RoboDK station: first test.rdk

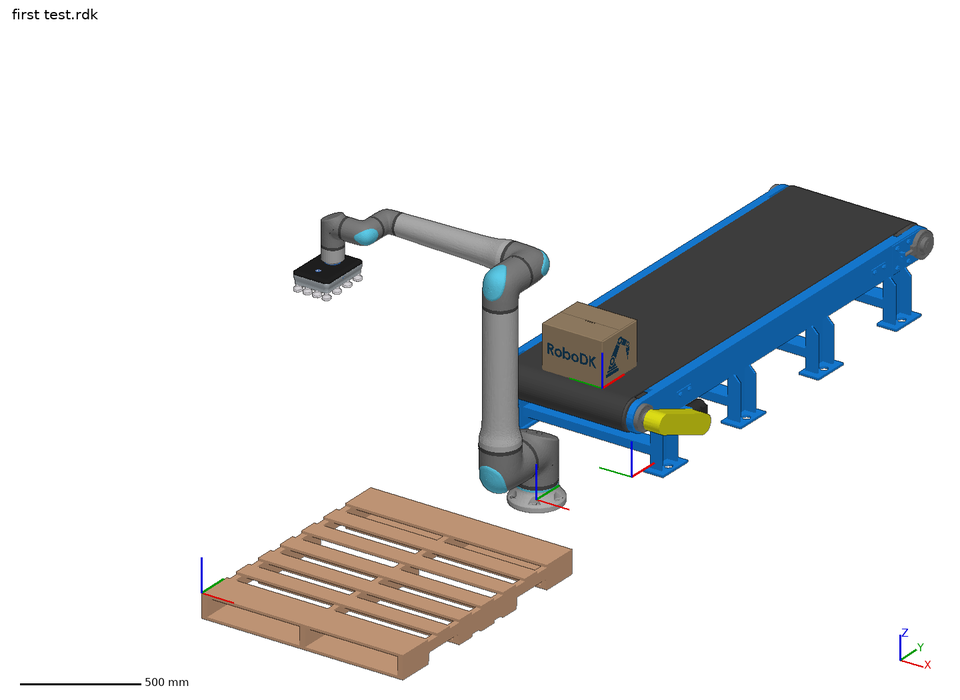
[picture v0: the station drawn from its stored meshes, robots at their saved joint values, targets as dots, program paths as lines]
Station first test (saved by RoboDK 5.9.2). Poses are relative to the parent item; angles as X-Y-Z fixed-axis rotations.
  - frame Conveyor Belt Wide (2m) Base at (200, 400, 0) mm, rotated rx 0 ry 0 rz 90 deg
    - robot Conveyor Belt Wide: 1 axes
        modified DH rows (alpha deg, a mm, theta deg, d mm): 0, 0, 0, 0 linear
        base shift (0, 0, 0) mm, rotated rx 0 ry 90 rz 0 deg
        joint limits [-900000] to [900000]; home [0]; saved at [0]
      - frame Box Center Pickup Point at (0, 150, 0) mm
        - object Box 12x10in (Closed) at (0, 0, 0) mm, size 252 x 305.4 x 216.7 mm, geometry from Box-12x10in-Closed.sld
  - frame Pallet Frame 40x48 at (-500, -1700, 110) mm
    - object Pallet 40x48in at (0, 0, 0) mm, size 1016 x 1219.2 x 114.3 mm, geometry from Pallet-40x48in.sld
  - frame UR20 Base at (0, 0, 0) mm
    - robot UR20: 6 axes
        modified DH rows (alpha deg, a mm, theta deg, d mm): 0, 0, 0, 236.2; 90, 0, -180, 0; 0, 861.8, 0, 0; 0, 727.7, 0, 201.9; -90, 0, 0, 159.4; 90, 0, 180, 154.8
        joint limits [-360, -360, -360, -360, -360, -360] to [360, 360, 360, 360, 360, 360]; home [0, -90, -90, 0, 90, 0]; saved at [0, -90, 90, -90, -90, 0]
      - tool OnRobot VGP20 Vacuum Gripper, TCP at (-36, 0, 106.49) mm, size 268.4 x 184.1 x 103.7 mm
